LIN {X 0,Y 130.457,Z 414.389,A -85,B 0,C 180,E1 -28269.621,E2 -28269.621} C_VEL
LIN {X 0,Y 125.281,Z 421.79,A -85,B 0,C 180,E1 -28270.976,E2 -28270.976} C_VEL
LIN {X 0,Y 118.932,Z 429.346,A -85,B 0,C 180,E1 -28272.835,E2 -28272.835} C_VEL
LIN {X 0,Y 111.008,Z 437.034,A -85,B 0,C 180,E1 -28275.509,E2 -28275.509} C_VEL
LIN {X 0,Y 103.666,Z 442.686,A -85,B 0,C 180,E1 -28278.357,E2 -28278.357} C_VEL
LIN {X 0,Y 97.893,Z 446.46,A -85,B 0,C 180,E1 -28281.046,E2 -28281.046} C_VEL
LIN {X 0,Y 92.339,Z 449.512,A -85,B 0,C 180,E1 -28284.033,E2 -28284.033} C_VEL
LIN {X 0,Y 87.083,Z 451.866,A -85,B 0,C 180,E1 -28287.41,E2 -28287.41} C_VEL
LIN {X 0,Y 82.167,Z 453.567,A -85,B 0,C 180,E1 -28291.205,E2 -28291.205} C_VEL
LIN {X 0,Y 77.631,Z 454.708,A -85,B 0,C 180,E1 -28295.437,E2 -28295.437} C_VEL
LIN {X 0,Y 71.023,Z 455.494,A -85,B 0,C 180,E1 -28303.815,E2 -28303.815} C_VEL
LIN {X 0,Y 67.098,Z 454.979,A -85,B 0,C 180,E1 -28311.065,E2 -28311.065} C_VEL
LIN {X 0,Y 64.842,Z 453.933,A -85,B 0,C 180,E1 -28317.186,E2 -28317.186} C_VEL
LIN {X 0,Y 62.895,Z 451.358,A -85,B 0,C 180,E1 -28326.979,E2 -28326.979} C_VEL
LIN {X 0,Y 62.503,Z 448.908,A -85,B 0,C 180,E1 -28333.675,E2 -28333.675} C_VEL
LIN {X 0,Y 63.308,Z 443.942,A -85,B 0,C 180,E1 -28343.628,E2 -28343.628} C_VEL
LIN {X 0,Y 65.146,Z 438.567,A -85,B 0,C 180,E1 -28351.547,E2 -28351.547} C_VEL
LIN {X 0,Y 67.153,Z 433.329,A -85,B 0,C 180,E1 -28357.518,E2 -28357.518} C_VEL
LIN {X 0,Y 69.776,Z 427.008,A -85,B 0,C 180,E1 -28363.1,E2 -28363.1} C_VEL
LIN {X 0,Y 72.514,Z 420.358,A -85,B 0,C 180,E1 -28367.631,E2 -28367.631} C_VEL
LIN {X 0,Y 75.671,Z 412.288,A -85,B 0,C 180,E1 -28371.809,E2 -28371.809} C_VEL
LIN {X 0,Y 78.693,Z 403.494,A -85,B 0,C 180,E1 -28375.219,E2 -28375.219} C_VEL
LIN {X 0,Y 81.712,Z 392.43,A -85,B 0,C 180,E1 -28378.324,E2 -28378.324} C_VEL
LIN {X 0,Y 83.873,Z 381.725,A -85,B 0,C 180,E1 -28380.297,E2 -28380.297} C_VEL
LIN {X 0,Y 85.27,Z 372.1,A -85,B 0,C 180,E1 -28381.419,E2 -28381.419} C_VEL
LIN {X 0,Y 87.182,Z 347.964,A -85,B 0,C 180,E1 -28383.17,E2 -28383.17} C_VEL
LIN {X 0,Y 84.324,Z 341.212,A -85,B 0,C 180,E1 -28385.816,E2 -28385.816} C_VEL
LIN {X 0,Y 79.131,Z 331.666,A -85,B 0,C 180,E1 -28391.138,E2 -28391.138} C_VEL
LIN {X 0,Y 75.765,Z 326.616,A -85,B 0,C 180,E1 -28395.162,E2 -28395.162} C_VEL
LIN {X 0,Y 73.243,Z 322.884,A -85,B 0,C 180,E1 -28398.715,E2 -28398.715} C_VEL
LIN {X 0,Y 70.889,Z 320.396,A -85,B 0,C 180,E1 -28402.421,E2 -28402.421} C_VEL
LIN {X 0,Y 69.816,Z 317.967,A -85,B 0,C 180,E1 -28404.656,E2 -28404.656} C_VEL
LIN {X 0,Y 67.219,Z 316.228,A -85,B 0,C 180,E1 -28410.108,E2 -28410.108} C_VEL
LIN {X 0,Y 65.712,Z 313.659,A -85,B 0,C 180,E1 -28414.906,E2 -28414.906} C_VEL
LIN {X 0,Y 65.448,Z 312.106,A -85,B 0,C 180,E1 -28416.696,E2 -28416.696} C_VEL
LIN {X 0,Y 70.33,Z 311.511,A -85,B 0,C 180,E1 -28437.877,E2 -28437.877} C_VEL
LIN {X 0,Y 75.148,Z 311.098,A -85,B 0,C 180,E1 -28444.711,E2 -28444.711} C_VEL
LIN {X 0,Y 80.078,Z 356.507,A -85,B 0,C 180,E1 -28453.675,E2 -28453.675} C_VEL
LIN {X 0,Y 81.204,Z 367.651,A -85,B 0,C 180,E1 -28456.127,E2 -28456.127} C_VEL
LIN {X 0,Y 81.915,Z 377.696,A -85,B 0,C 180,E1 -28459.031,E2 -28459.031} C_VEL
LIN {X 0,Y 82.52,Z 385.251,A -85,B 0,C 180,E1 -28461.893,E2 -28461.893} C_VEL
LIN {X 0,Y 83.392,Z 393.266,A -85,B 0,C 180,E1 -28465.969,E2 -28465.969} C_VEL
LIN {X 0,Y 84.869,Z 401.147,A -85,B 0,C 180,E1 -28470.72,E2 -28470.72} C_VEL
LIN {X 0,Y 87.441,Z 409.064,A -85,B 0,C 180,E1 -28475.939,E2 -28475.939} C_VEL
LIN {X 0,Y 93.038,Z 419.345,A -85,B 0,C 180,E1 -28482.849,E2 -28482.849} C_VEL
LIN {X 0,Y 94.672,Z 421.602,A -85,B 0,C 180,E1 -28484.351,E2 -28484.351} C_VEL
LIN {X 0,Y 93.114,Z 419.795,A -85,B 0,C 180,E1 -28487.21,E2 -28487.21} C_VEL
LIN {X 0,Y 88.882,Z 413.219,A -85,B 0,C 180,E1 -28493.557,E2 -28493.557} C_VEL
LIN {X 0,Y 84.438,Z 418.04,A -85,B 0,C 180,E1 -28494.363,E2 -28494.363} C_VEL
LIN {X 0,Y 79.435,Z 424.487,A -85,B 0,C 180,E1 -28496.428,E2 -28496.428} C_VEL
LIN {X 0,Y 74.169,Z 431.806,A -85,B 0,C 180,E1 -28500.166,E2 -28500.166} C_VEL
LIN {X 0,Y 70.273,Z 437.549,A -85,B 0,C 180,E1 -28504.351,E2 -28504.351} C_VEL
LIN {X 0,Y 66.983,Z 443.216,A -85,B 0,C 180,E1 -28510.061,E2 -28510.061} C_VEL
LIN {X 0,Y 64.441,Z 448.562,A -85,B 0,C 180,E1 -28517.4,E2 -28517.4} C_VEL
LIN {X 0,Y 63.41,Z 452.058,A -85,B 0,C 180,E1 -28523.635,E2 -28523.635} C_VEL
LIN {X 0,Y 63.272,Z 454.934,A -85,B 0,C 180,E1 -28529.999,E2 -28529.999} C_VEL
LIN {X 0,Y 63.085,Z 457.125,A -85,B 0,C 180,E1 -28536.395,E2 -28536.395} C_VEL
LIN {X 0,Y 63.598,Z 458.696,A -85,B 0,C 180,E1 -28542.767,E2 -28542.767} C_VEL
LIN {X 0,Y 64.839,Z 459.786,A -85,B 0,C 180,E1 -28548.975,E2 -28548.975} C_VEL
LIN {X 0,Y 66.817,Z 460.43,A -85,B 0,C 180,E1 -28554.879,E2 -28554.879} C_VEL
LIN {X 0,Y 69.423,Z 460.623,A -85,B 0,C 180,E1 -28560.408,E2 -28560.408} C_VEL
LIN {X 0,Y 72.698,Z 460.247,A -85,B 0,C 180,E1 -28565.452,E2 -28565.452} C_VEL
LIN {X 0,Y 76.592,Z 459.396,A -85,B 0,C 180,E1 -28569.963,E2 -28569.963} C_VEL
LIN {X 0,Y 80.924,Z 458.092,A -85,B 0,C 180,E1 -28574.008,E2 -28574.008} C_VEL
LIN {X 0,Y 88.109,Z 455.143,A -85,B 0,C 180,E1 -28579.267,E2 -28579.267} C_VEL
LIN {X 0,Y 93.327,Z 452.493,A -85,B 0,C 180,E1 -28582.25,E2 -28582.25} C_VEL
LIN {X 0,Y 101.608,Z 447.322,A -85,B 0,C 180,E1 -28586.099,E2 -28586.099} C_VEL
LIN {X 0,Y 109.921,Z 440.844,A -85,B 0,C 180,E1 -28589.31,E2 -28589.31} C_VEL
LIN {X 0,Y 117.751,Z 433.257,A -85,B 0,C 180,E1 -28591.685,E2 -28591.685} C_VEL
LIN {X 0,Y 123.906,Z 426.049,A -85,B 0,C 180,E1 -28593.296,E2 -28593.296} C_VEL
LIN {X 0,Y 129.407,Z 418.363,A -85,B 0,C 180,E1 -28594.54,E2 -28594.54} C_VEL
LIN {X 0,Y 133.967,Z 410.731,A -85,B 0,C 180,E1 -28595.444,E2 -28595.444} C_VEL
LIN {X 0,Y 138.255,Z 401.917,A -85,B 0,C 180,E1 -28596.205,E2 -28596.205} C_VEL
LIN {X 0,Y 139.851,Z 398.143,A -85,B 0,C 180,E1 -28596.509,E2 -28596.509} C_VEL
LIN {X 0,Y 139.681,Z 393.765,A -85,B 0,C 180,E1 -28599.369,E2 -28599.369} C_VEL
LIN {X 0,Y 139.428,Z 392.17,A -85,B 0,C 180,E1 -28600.927,E2 -28600.927} C_VEL
LIN {X 0,Y 138.957,Z 389.849,A -85,B 0,C 180,E1 -28603.935,E2 -28603.935} C_VEL
LIN {X 0,Y 138.331,Z 386.897,A -85,B 0,C 180,E1 -28611.224,E2 -28611.224} C_VEL
LIN {X 0,Y 138.451,Z 386.702,A -85,B 0,C 180,E1 -28614.164,E2 -28614.164} C_VEL
LIN {X 0,Y 138.714,Z 389.539,A -85,B 0,C 180,E1 -28619.991,E2 -28619.991} C_VEL
LIN {X 0,Y 139.208,Z 393.208,A -85,B 0,C 180,E1 -28624.334,E2 -28624.334} C_VEL
LIN {X 0,Y 139.334,Z 394.063,A -85,B 0,C 180,E1 -28625.176,E2 -28625.176} C_VEL
LIN {X 0,Y 139.116,Z 395.586,A -85,B 0,C 180,E1 -28625.911,E2 -28625.911} C_VEL
LIN {X 0,Y 138.136,Z 398.315,A -85,B 0,C 180,E1 -28626.389,E2 -28626.389} C_VEL
LIN {X 0,Y 136.101,Z 402.524,A -85,B 0,C 180,E1 -28626.493,E2 -28626.493} C_VEL
LIN {X 0,Y 131.283,Z 410.331,A -85,B 0,C 180,E1 -28626.163,E2 -28626.163} C_VEL
LIN {X 0,Y 129.637,Z 412.827,A -85,B 0,C 180,E1 -28626.35,E2 -28626.35} C_VEL
LIN {X 0,Y 124.077,Z 420.81,A -85,B 0,C 180,E1 -28627.595,E2 -28627.595} C_VEL
LIN {X 0,Y 119.137,Z 426.82,A -85,B 0,C 180,E1 -28628.854,E2 -28628.854} C_VEL
LIN {X 0,Y 112.163,Z 433.882,A -85,B 0,C 180,E1 -28630.823,E2 -28630.823} C_VEL
LIN {X 0,Y 104.693,Z 440.112,A -85,B 0,C 180,E1 -28633.254,E2 -28633.254} C_VEL
LIN {X 0,Y 98.493,Z 444.382,A -85,B 0,C 180,E1 -28635.575,E2 -28635.575} C_VEL
LIN {X 0,Y 92.028,Z 448.107,A -85,B 0,C 180,E1 -28638.443,E2 -28638.443} C_VEL
LIN {X 0,Y 83.908,Z 451.828,A -85,B 0,C 180,E1 -28642.879,E2 -28642.879} C_VEL
LIN {X 0,Y 78.468,Z 453.66,A -85,B 0,C 180,E1 -28646.585,E2 -28646.585} C_VEL
LIN {X 0,Y 73.547,Z 454.886,A -85,B 0,C 180,E1 -28650.684,E2 -28650.684} C_VEL
LIN {X 0,Y 68.987,Z 455.606,A -85,B 0,C 180,E1 -28655.415,E2 -28655.415} C_VEL
LIN {X 0,Y 64.945,Z 455.807,A -85,B 0,C 180,E1 -28660.758,E2 -28660.758} C_VEL
LIN {X 0,Y 61.48,Z 455.417,A -85,B 0,C 180,E1 -28666.696,E2 -28666.696} C_VEL
LIN {X 0,Y 58.722,Z 454.44,A -85,B 0,C 180,E1 -28673.245,E2 -28673.245} C_VEL
LIN {X 0,Y 56.128,Z 452.049,A -85,B 0,C 180,E1 -28684.009,E2 -28684.009} C_VEL
LIN {X 0,Y 55.418,Z 448.224,A -85,B 0,C 180,E1 -28695.309,E2 -28695.309} C_VEL
LIN {X 0,Y 56.395,Z 443.599,A -85,B 0,C 180,E1 -28705.23,E2 -28705.23} C_VEL
LIN {X 0,Y 58.367,Z 438.473,A -85,B 0,C 180,E1 -28713.453,E2 -28713.453} C_VEL
LIN {X 0,Y 60.615,Z 433.152,A -85,B 0,C 180,E1 -28720.017,E2 -28720.017} C_VEL
LIN {X 0,Y 63.546,Z 426.73,A -85,B 0,C 180,E1 -28726.052,E2 -28726.052} C_VEL
LIN {X 0,Y 67.556,Z 417.869,A -85,B 0,C 180,E1 -28732.156,E2 -28732.156} C_VEL
LIN {X 0,Y 71.497,Z 407.795,A -85,B 0,C 180,E1 -28736.947,E2 -28736.947} C_VEL
LIN {X 0,Y 74.353,Z 399.47,A -85,B 0,C 180,E1 -28739.753,E2 -28739.753} C_VEL
LIN {X 0,Y 76.853,Z 390.146,A -85,B 0,C 180,E1 -28742.111,E2 -28742.111} C_VEL
LIN {X 0,Y 78.787,Z 380.756,A -85,B 0,C 180,E1 -28743.772,E2 -28743.772} C_VEL
LIN {X 0,Y 80.185,Z 371.132,A -85,B 0,C 180,E1 -28744.848,E2 -28744.848} C_VEL
LIN {X 0,Y 81.93,Z 350.008,A -85,B 0,C 180,E1 -28746.413,E2 -28746.413} C_VEL
LIN {X 0,Y 79.46,Z 344.241,A -85,B 0,C 180,E1 -28749.083,E2 -28749.083} C_VEL
LIN {X 0,Y 75.348,Z 336.338,A -85,B 0,C 180,E1 -28754.021,E2 -28754.021} C_VEL
LIN {X 0,Y 72.573,Z 332.018,A -85,B 0,C 180,E1 -28757.856,E2 -28757.856} C_VEL
LIN {X 0,Y 70.65,Z 329.013,A -85,B 0,C 180,E1 -28760.957,E2 -28760.957} C_VEL
LIN {X 0,Y 68.282,Z 325.962,A -85,B 0,C 180,E1 -28765.357,E2 -28765.357} C_VEL
LIN {X 0,Y 67.655,Z 324.536,A -85,B 0,C 180,E1 -28766.865,E2 -28766.865} C_VEL
LIN {X 0,Y 65.267,Z 322.375,A -85,B 0,C 180,E1 -28772.878,E2 -28772.878} C_VEL
LIN {X 0,Y 64.053,Z 319.715,A -85,B 0,C 180,E1 -28777.864,E2 -28777.864} C_VEL
LIN {X 0,Y 63.854,Z 318.969,A -85,B 0,C 180,E1 -28779.063,E2 -28779.063} C_VEL
LIN {X 0,Y 62.674,Z 317.487,A -85,B 0,C 180,E1 -28789.522,E2 -28789.522} C_VEL
LIN {X 0,Y 63.268,Z 315.101,A -85,B 0,C 180,E1 -28796.991,E2 -28796.991} C_VEL
LIN {X 0,Y 64.046,Z 312.858,A -85,B 0,C 180,E1 -28800.413,E2 -28800.413} C_VEL
LIN {X 0,Y 64.388,Z 312.272,A -85,B 0,C 180,E1 -28801.193,E2 -28801.193} C_VEL
LIN {X 0,Y 70.156,Z 311.553,A -85,B 0,C 180,E1 -28808.661,E2 -28808.661} C_VEL
LIN {X 0,Y 75.977,Z 356.93,A -85,B 0,C 180,E1 -28818.034,E2 -28818.034} C_VEL
LIN {X 0,Y 77.242,Z 367.844,A -85,B 0,C 180,E1 -28820.612,E2 -28820.612} C_VEL
LIN {X 0,Y 78.05,Z 376.177,A -85,B 0,C 180,E1 -28823.217,E2 -28823.217} C_VEL
LIN {X 0,Y 78.768,Z 382.764,A -85,B 0,C 180,E1 -28825.801,E2 -28825.801} C_VEL
LIN {X 0,Y 80.176,Z 392.373,A -85,B 0,C 180,E1 -28830.941,E2 -28830.941} C_VEL
LIN {X 0,Y 82.567,Z 401.252,A -85,B 0,C 180,E1 -28836.59,E2 -28836.59} C_VEL
LIN {X 0,Y 87.688,Z 412.169,A -85,B 0,C 180,E1 -28843.834,E2 -28843.834} C_VEL
LIN {X 0,Y 89.092,Z 414.368,A -85,B 0,C 180,E1 -28845.25,E2 -28845.25} C_VEL
LIN {X 0,Y 85.771,Z 408.902,A -85,B 0,C 180,E1 -28850.45,E2 -28850.45} C_VEL
LIN {X 0,Y 81.591,Z 413.122,A -85,B 0,C 180,E1 -28850.849,E2 -28850.849} C_VEL
LIN {X 0,Y 77.065,Z 418.627,A -85,B 0,C 180,E1 -28852.005,E2 -28852.005} C_VEL
LIN {X 0,Y 72.249,Z 424.988,A -85,B 0,C 180,E1 -28854.291,E2 -28854.291} C_VEL
LIN {X 0,Y 66.949,Z 432.195,A -85,B 0,C 180,E1 -28858.338,E2 -28858.338} C_VEL
LIN {X 0,Y 63.263,Z 437.614,A -85,B 0,C 180,E1 -28862.755,E2 -28862.755} C_VEL
LIN {X 0,Y 59.702,Z 443.409,A -85,B 0,C 180,E1 -28869.318,E2 -28869.318} C_VEL
LIN {X 0,Y 57.58,Z 447.722,A -85,B 0,C 180,E1 -28875.869,E2 -28875.869} C_VEL
LIN {X 0,Y 56.195,Z 452.827,A -85,B 0,C 180,E1 -28886.413,E2 -28886.413} C_VEL
LIN {X 0,Y 56.205,Z 454.283,A -85,B 0,C 180,E1 -28889.999,E2 -28889.999} C_VEL
LIN {X 0,Y 56.055,Z 456.497,A -85,B 0,C 180,E1 -28897.201,E2 -28897.201} C_VEL
LIN {X 0,Y 56.695,Z 458.149,A -85,B 0,C 180,E1 -28904.353,E2 -28904.353} C_VEL
LIN {X 0,Y 58.16,Z 459.327,A -85,B 0,C 180,E1 -28911.254,E2 -28911.254} C_VEL
LIN {X 0,Y 60.43,Z 460.057,A -85,B 0,C 180,E1 -28917.722,E2 -28917.722} C_VEL
LIN {X 0,Y 63.382,Z 460.289,A -85,B 0,C 180,E1 -28923.669,E2 -28923.669} C_VEL
LIN {X 0,Y 67.041,Z 459.963,A -85,B 0,C 180,E1 -28928.974,E2 -28928.974} C_VEL
LIN {X 0,Y 71.296,Z 459.199,A -85,B 0,C 180,E1 -28933.631,E2 -28933.631} C_VEL
LIN {X 0,Y 75.966,Z 457.983,A -85,B 0,C 180,E1 -28937.74,E2 -28937.74} C_VEL
LIN {X 0,Y 83.656,Z 455.131,A -85,B 0,C 180,E1 -28942.948,E2 -28942.948} C_VEL
LIN {X 0,Y 92.002,Z 451.056,A -85,B 0,C 180,E1 -28947.169,E2 -28947.169} C_VEL
LIN {X 0,Y 100.766,Z 445.605,A -85,B 0,C 180,E1 -28950.67,E2 -28950.67} C_VEL
LIN {X 0,Y 108.352,Z 439.686,A -85,B 0,C 180,E1 -28953.107,E2 -28953.107} C_VEL
LIN {X 0,Y 116.145,Z 432.213,A -85,B 0,C 180,E1 -28955.182,E2 -28955.182} C_VEL
LIN {X 0,Y 122.5,Z 424.864,A -85,B 0,C 180,E1 -28956.626,E2 -28956.626} C_VEL
LIN {X 0,Y 128.153,Z 417.003,A -85,B 0,C 180,E1 -28957.732,E2 -28957.732} C_VEL
LIN {X 0,Y 133.325,Z 408.252,A -85,B 0,C 180,E1 -28958.596,E2 -28958.596} C_VEL
LIN {X 0,Y 136.379,Z 401.889,A -85,B 0,C 180,E1 -28959.07,E2 -28959.07} C_VEL
LIN {X 0,Y 136.676,Z 399.651,A -85,B 0,C 180,E1 -28960.463,E2 -28960.463} C_VEL
LIN {X 0,Y 136.418,Z 397.023,A -85,B 0,C 180,E1 -28963.627,E2 -28963.627} C_VEL
LIN {X 0,Y 136.274,Z 396.091,A -85,B 0,C 180,E1 -28965.047,E2 -28965.047} C_VEL
LIN {X 0,Y 135.969,Z 393.72,A -85,B 0,C 180,E1 -28971.07,E2 -28971.07} C_VEL
LIN {X 0,Y 136.066,Z 393.495,A -85,B 0,C 180,E1 -28974.061,E2 -28974.061} C_VEL
LIN {X 0,Y 136.064,Z 396.477,A -85,B 0,C 180,E1 -28979.99,E2 -28979.99} C_VEL
LIN {X 0,Y 136.138,Z 400.277,A -85,B 0,C 180,E1 -28984.58,E2 -28984.58} C_VEL
LIN {X 0,Y 136.146,Z 400.62,A -85,B 0,C 180,E1 -28984.913,E2 -28984.913} C_VEL
LIN {X 0,Y 131.331,Z 410.103,A -85,B 0,C 180,E1 -28985.99,E2 -28985.99} C_VEL
LIN {X 0,Y 129.637,Z 412.827,A -85,B 0,C 180,E1 -28986.35,E2 -28986.35} C_VEL
LIN {X 0,Y 126.256,Z 417.745,A -85,B 0,C 180,E1 -28986.767,E2 -28986.767} C_VEL
LIN {X 0,Y 119.636,Z 425.325,A -85,B 0,C 180,E1 -28986.795,E2 -28986.795} C_VEL
LIN {X 0,Y 112.539,Z 432.075,A -85,B 0,C 180,E1 -28987.002,E2 -28987.002} C_VEL
LIN {X 0,Y 108.327,Z 435.68,A -85,B 0,C 180,E1 -28987.775,E2 -28987.775} C_VEL
LIN {X 0,Y 99.979,Z 442.094,A -85,B 0,C 180,E1 -28990.226,E2 -28990.226} C_VEL
LIN {X 0,Y 91.444,Z 447.21,A -85,B 0,C 180,E1 -28993.315,E2 -28993.315} C_VEL
LIN {X 0,Y 84.276,Z 450.622,A -85,B 0,C 180,E1 -28996.462,E2 -28996.462} C_VEL
LIN {X 0,Y 74.432,Z 454.03,A -85,B 0,C 180,E1 -29002.171,E2 -29002.171} C_VEL
LIN {X 0,Y 70.021,Z 455.074,A -85,B 0,C 180,E1 -29005.404,E2 -29005.404} C_VEL
LIN {X 0,Y 64.941,Z 455.898,A -85,B 0,C 180,E1 -29010.031,E2 -29010.031} C_VEL
LIN {X 0,Y 59.94,Z 456.158,A -85,B 0,C 180,E1 -29015.863,E2 -29015.863} C_VEL
LIN {X 0,Y 56.28,Z 455.815,A -85,B 0,C 180,E1 -29021.476,E2 -29021.476} C_VEL
LIN {X 0,Y 52.936,Z 454.945,A -85,B 0,C 180,E1 -29028.41,E2 -29028.41} C_VEL
LIN {X 0,Y 50.205,Z 453.344,A -85,B 0,C 180,E1 -29037.081,E2 -29037.081} C_VEL
LIN {X 0,Y 48.504,Z 450.38,A -85,B 0,C 180,E1 -29048.764,E2 -29048.764} C_VEL
LIN {X 0,Y 48.755,Z 445.867,A -85,B 0,C 180,E1 -29061.714,E2 -29061.714} C_VEL
LIN {X 0,Y 50.576,Z 440.812,A -85,B 0,C 180,E1 -29071.992,E2 -29071.992} C_VEL
LIN {X 0,Y 53.542,Z 434.424,A -85,B 0,C 180,E1 -29081.357,E2 -29081.357} C_VEL
LIN {X 0,Y 56.637,Z 428.197,A -85,B 0,C 180,E1 -29088.074,E2 -29088.074} C_VEL
LIN {X 0,Y 59.938,Z 421.64,A -85,B 0,C 180,E1 -29093.313,E2 -29093.313} C_VEL
LIN {X 0,Y 63.183,Z 414.694,A -85,B 0,C 180,E1 -29097.502,E2 -29097.502} C_VEL
LIN {X 0,Y 66.232,Z 407.319,A -85,B 0,C 180,E1 -29100.892,E2 -29100.892} C_VEL
LIN {X 0,Y 68.817,Z 400.372,A -85,B 0,C 180,E1 -29103.295,E2 -29103.295} C_VEL
LIN {X 0,Y 71.465,Z 391.239,A -85,B 0,C 180,E1 -29105.727,E2 -29105.727} C_VEL
LIN {X 0,Y 73.636,Z 381.781,A -85,B 0,C 180,E1 -29107.434,E2 -29107.434} C_VEL
LIN {X 0,Y 75.176,Z 372.245,A -85,B 0,C 180,E1 -29108.529,E2 -29108.529} C_VEL
LIN {X 0,Y 76.972,Z 352.143,A -85,B 0,C 180,E1 -29110.079,E2 -29110.079} C_VEL
LIN {X 0,Y 73.015,Z 343.412,A -85,B 0,C 180,E1 -29115.331,E2 -29115.331} C_VEL
LIN {X 0,Y 69.63,Z 337.529,A -85,B 0,C 180,E1 -29120.639,E2 -29120.639} C_VEL
LIN {X 0,Y 68.047,Z 334.961,A -85,B 0,C 180,E1 -29123.6,E2 -29123.6} C_VEL
LIN {X 0,Y 65.774,Z 331.311,A -85,B 0,C 180,E1 -29128.778,E2 -29128.778} C_VEL
LIN {X 0,Y 63.04,Z 327.611,A -85,B 0,C 180,E1 -29137.813,E2 -29137.813} C_VEL
LIN {X 0,Y 62.539,Z 325.828,A -85,B 0,C 180,E1 -29141.11,E2 -29141.11} C_VEL
LIN {X 0,Y 61.815,Z 324.122,A -85,B 0,C 180,E1 -29151.851,E2 -29151.851} C_VEL
LIN {X 0,Y 62.803,Z 321.557,A -85,B 0,C 180,E1 -29159.64,E2 -29159.64} C_VEL
LIN {X 0,Y 64.008,Z 319.003,A -85,B 0,C 180,E1 -29163.953,E2 -29163.953} C_VEL
LIN {X 0,Y 64.879,Z 318.49,A -85,B 0,C 180,E1 -29166.824,E2 -29166.824} C_VEL
LIN {X 0,Y 65.14,Z 329.275,A -85,B 0,C 180,E1 -29171.494,E2 -29171.494} C_VEL
LIN {X 0,Y 65.779,Z 333.915,A -85,B 0,C 180,E1 -29174.316,E2 -29174.316} C_VEL
LIN {X 0,Y 66.257,Z 335.047,A -85,B 0,C 180,E1 -29175.582,E2 -29175.582} C_VEL
LIN {X 0,Y 66.769,Z 334.861,A -85,B 0,C 180,E1 -29176.494,E2 -29176.494} C_VEL
LIN {X 0,Y 67.367,Z 332.904,A -85,B 0,C 180,E1 -29177.078,E2 -29177.078} C_VEL
LIN {X 0,Y 67.851,Z 329.395,A -85,B 0,C 180,E1 -29177.062,E2 -29177.062} C_VEL
LIN {X 0,Y 72.311,Z 356.278,A -85,B 0,C 180,E1 -29182.734,E2 -29182.734} C_VEL
LIN {X 0,Y 73.954,Z 367.504,A -85,B 0,C 180,E1 -29185.525,E2 -29185.525} C_VEL
LIN {X 0,Y 75.118,Z 376.804,A -85,B 0,C 180,E1 -29188.671,E2 -29188.671} C_VEL
LIN {X 0,Y 76.088,Z 384.013,A -85,B 0,C 180,E1 -29192.099,E2 -29192.099} C_VEL
LIN {X 0,Y 78.185,Z 392.918,A -85,B 0,C 180,E1 -29197.373,E2 -29197.373} C_VEL
LIN {X 0,Y 82.43,Z 403.63,A -85,B 0,C 180,E1 -29204.39,E2 -29204.39} C_VEL
LIN {X 0,Y 83.1,Z 404.894,A -85,B 0,C 180,E1 -29205.192,E2 -29205.192} C_VEL
LIN {X 0,Y 82.699,Z 404.297,A -85,B 0,C 180,E1 -29207.429,E2 -29207.429} C_VEL
LIN {X 0,Y 78.275,Z 408.962,A -85,B 0,C 180,E1 -29207.337,E2 -29207.337} C_VEL
LIN {X 0,Y 72.631,Z 415.885,A -85,B 0,C 180,E1 -29208.297,E2 -29208.297} C_VEL
LIN {X 0,Y 66.736,Z 423.585,A -85,B 0,C 180,E1 -29210.811,E2 -29210.811} C_VEL
LIN {X 0,Y 61.108,Z 430.962,A -85,B 0,C 180,E1 -29214.896,E2 -29214.896} C_VEL
LIN {X 0,Y 56.642,Z 437.197,A -85,B 0,C 180,E1 -29220.242,E2 -29220.242} C_VEL
LIN {X 0,Y 53.184,Z 442.454,A -85,B 0,C 180,E1 -29226.643,E2 -29226.643} C_VEL
LIN {X 0,Y 50.762,Z 446.88,A -85,B 0,C 180,E1 -29233.923,E2 -29233.923} C_VEL
LIN {X 0,Y 49.393,Z 450.583,A -85,B 0,C 180,E1 -29241.818,E2 -29241.818} C_VEL
LIN {X 0,Y 49.127,Z 453.589,A -85,B 0,C 180,E1 -29249.998,E2 -29249.998} C_VEL
LIN {X 0,Y 49.054,Z 455.86,A -85,B 0,C 180,E1 -29258.236,E2 -29258.236} C_VEL
LIN {X 0,Y 49.858,Z 457.603,A -85,B 0,C 180,E1 -29266.373,E2 -29266.373} C_VEL
LIN {X 0,Y 51.604,Z 458.869,A -85,B 0,C 180,E1 -29274.114,E2 -29274.114} C_VEL
LIN {X 0,Y 54.232,Z 459.679,A -85,B 0,C 180,E1 -29281.221,E2 -29281.221} C_VEL
LIN {X 0,Y 57.592,Z 459.921,A -85,B 0,C 180,E1 -29287.599,E2 -29287.599} C_VEL
LIN {X 0,Y 61.687,Z 459.68,A -85,B 0,C 180,E1 -29293.123,E2 -29293.123} C_VEL
LIN {X 0,Y 66.339,Z 459.008,A -85,B 0,C 180,E1 -29297.865,E2 -29297.865} C_VEL
LIN {X 0,Y 71.376,Z 457.888,A -85,B 0,C 180,E1 -29301.971,E2 -29301.971} C_VEL
LIN {X 0,Y 79.588,Z 455.138,A -85,B 0,C 180,E1 -29307.022,E2 -29307.022} C_VEL
LIN {X 0,Y 88.353,Z 451.169,A -85,B 0,C 180,E1 -29311.042,E2 -29311.042} C_VEL
LIN {X 0,Y 94.433,Z 447.762,A -85,B 0,C 180,E1 -29313.261,E2 -29313.261} C_VEL
LIN {X 0,Y 102.166,Z 442.495,A -85,B 0,C 180,E1 -29315.707,E2 -29315.707} C_VEL
LIN {X 0,Y 108.538,Z 437.345,A -85,B 0,C 180,E1 -29317.324,E2 -29317.324} C_VEL
LIN {X 0,Y 114.974,Z 431.172,A -85,B 0,C 180,E1 -29318.776,E2 -29318.776} C_VEL
LIN {X 0,Y 120.691,Z 424.698,A -85,B 0,C 180,E1 -29319.88,E2 -29319.88} C_VEL
LIN {X 0,Y 126.482,Z 416.867,A -85,B 0,C 180,E1 -29320.839,E2 -29320.839} C_VEL
LIN {X 0,Y 131.793,Z 408.081,A -85,B 0,C 180,E1 -29321.598,E2 -29321.598} C_VEL
LIN {X 0,Y 133.189,Z 405.532,A -85,B 0,C 180,E1 -29321.769,E2 -29321.769} C_VEL
LIN {X 0,Y 133.336,Z 404.016,A -85,B 0,C 180,E1 -29323.137,E2 -29323.137} C_VEL
LIN {X 0,Y 133.273,Z 402.921,A -85,B 0,C 180,E1 -29324.703,E2 -29324.703} C_VEL
LIN {X 0,Y 133.129,Z 400.436,A -85,B 0,C 180,E1 -29330.878,E2 -29330.878} C_VEL
LIN {X 0,Y 133.25,Z 400.082,A -85,B 0,C 180,E1 -29333.935,E2 -29333.935} C_VEL
LIN {X 0,Y 132.908,Z 403.136,A -85,B 0,C 180,E1 -29339.99,E2 -29339.99} C_VEL
LIN {X 0,Y 132.744,Z 404.85,A -85,B 0,C 180,E1 -29342.267,E2 -29342.267} C_VEL
LIN {X 0,Y 131.255,Z 407.626,A -85,B 0,C 180,E1 -29342.664,E2 -29342.664} C_VEL
LIN {X 0,Y 125.882,Z 416.262,A -85,B 0,C 180,E1 -29343.664,E2 -29343.664} C_VEL
LIN {X 0,Y 119.919,Z 424.086,A -85,B 0,C 180,E1 -29344.931,E2 -29344.931} C_VEL
LIN {X 0,Y 113.176,Z 431.347,A -85,B 0,C 180,E1 -29346.507,E2 -29346.507} C_VEL
LIN {X 0,Y 108.327,Z 435.68,A -85,B 0,C 180,E1 -29347.775,E2 -29347.775} C_VEL
LIN {X 0,Y 105.283,Z 438.116,A -85,B 0,C 180,E1 -29348.246,E2 -29348.246} C_VEL
LIN {X 0,Y 99.597,Z 441.771,A -85,B 0,C 180,E1 -29348.102,E2 -29348.102} C_VEL
LIN {X 0,Y 93.677,Z 445.056,A -85,B 0,C 180,E1 -29347.983,E2 -29347.983} C_VEL
LIN {X 0,Y 90.269,Z 446.858,A -85,B 0,C 180,E1 -29348.611,E2 -29348.611} C_VEL
LIN {X 0,Y 82.478,Z 450.591,A -85,B 0,C 180,E1 -29351.506,E2 -29351.506} C_VEL
LIN {X 0,Y 73.109,Z 453.797,A -85,B 0,C 180,E1 -29355.994,E2 -29355.994} C_VEL
LIN {X 0,Y 67.161,Z 455.26,A -85,B 0,C 180,E1 -29359.648,E2 -29359.648} C_VEL
LIN {X 0,Y 61.535,Z 456.172,A -85,B 0,C 180,E1 -29363.982,E2 -29363.982} C_VEL
LIN {X 0,Y 54.94,Z 456.487,A -85,B 0,C 180,E1 -29370.748,E2 -29370.748} C_VEL
LIN {X 0,Y 47.621,Z 455.443,A -85,B 0,C 180,E1 -29382.449,E2 -29382.449} C_VEL
LIN {X 0,Y 43.684,Z 453.627,A -85,B 0,C 180,E1 -29393.5,E2 -29393.5} C_VEL
LIN {X 0,Y 41.684,Z 451.092,A -85,B 0,C 180,E1 -29405.073,E2 -29405.073} C_VEL
LIN {X 0,Y 41.228,Z 448.311,A -85,B 0,C 180,E1 -29415.187,E2 -29415.187} C_VEL
LIN {X 0,Y 42.208,Z 444.199,A -85,B 0,C 180,E1 -29426.835,E2 -29426.835} C_VEL
LIN {X 0,Y 44.435,Z 439.471,A -85,B 0,C 180,E1 -29436.814,E2 -29436.814} C_VEL
LIN {X 0,Y 47.236,Z 434.214,A -85,B 0,C 180,E1 -29445.094,E2 -29445.094} C_VEL
LIN {X 0,Y 50.778,Z 427.882,A -85,B 0,C 180,E1 -29452.374,E2 -29452.374} C_VEL
LIN {X 0,Y 54.467,Z 421.205,A -85,B 0,C 180,E1 -29457.889,E2 -29457.889} C_VEL
LIN {X 0,Y 58.505,Z 413.184,A -85,B 0,C 180,E1 -29462.672,E2 -29462.672} C_VEL
LIN {X 0,Y 62.963,Z 402.986,A -85,B 0,C 180,E1 -29466.869,E2 -29466.869} C_VEL
LIN {X 0,Y 66.498,Z 392.073,A -85,B 0,C 180,E1 -29469.904,E2 -29469.904} C_VEL
LIN {X 0,Y 68.919,Z 382.191,A -85,B 0,C 180,E1 -29471.711,E2 -29471.711} C_VEL
LIN {X 0,Y 70.6,Z 372.517,A -85,B 0,C 180,E1 -29472.784,E2 -29472.784} C_VEL
LIN {X 0,Y 72.342,Z 354.689,A -85,B 0,C 180,E1 -29474.153,E2 -29474.153} C_VEL
LIN {X 0,Y 69.012,Z 346.993,A -85,B 0,C 180,E1 -29479.561,E2 -29479.561} C_VEL
LIN {X 0,Y 65.986,Z 341.335,A -85,B 0,C 180,E1 -29485.61,E2 -29485.61} C_VEL
LIN {X 0,Y 63.597,Z 337.346,A -85,B 0,C 180,E1 -29492.001,E2 -29492.001} C_VEL
LIN {X 0,Y 61.628,Z 333.965,A -85,B 0,C 180,E1 -29500.419,E2 -29500.419} C_VEL
LIN {X 0,Y 61.324,Z 332.692,A -85,B 0,C 180,E1 -29503.118,E2 -29503.118} C_VEL
LIN {X 0,Y 61.058,Z 330.786,A -85,B 0,C 180,E1 -29514.251,E2 -29514.251} C_VEL
LIN {X 0,Y 62.468,Z 328.005,A -85,B 0,C 180,E1 -29522.311,E2 -29522.311} C_VEL
LIN {X 0,Y 62.866,Z 327.318,A -85,B 0,C 180,E1 -29523.69,E2 -29523.69} C_VEL
LIN {X 0,Y 62.997,Z 335.729,A -85,B 0,C 180,E1 -29528.037,E2 -29528.037} C_VEL
LIN {X 0,Y 63.702,Z 340.13,A -85,B 0,C 180,E1 -29531.555,E2 -29531.555} C_VEL
LIN {X 0,Y 64.717,Z 341.838,A -85,B 0,C 180,E1 -29534.373,E2 -29534.373} C_VEL
LIN {X 0,Y 65.051,Z 342.168,A -85,B 0,C 180,E1 -29535.15,E2 -29535.15} C_VEL
LIN {X 0,Y 66.24,Z 361.269,A -85,B 0,C 180,E1 -29541.819,E2 -29541.819} C_VEL
LIN {X 0,Y 68.211,Z 378.087,A -85,B 0,C 180,E1 -29548.017,E2 -29548.017} C_VEL
LIN {X 0,Y 69.235,Z 385.547,A -85,B 0,C 180,E1 -29551.369,E2 -29551.369} C_VEL
LIN {X 0,Y 70.865,Z 393.104,A -85,B 0,C 180,E1 -29555.658,E2 -29555.658} C_VEL
LIN {X 0,Y 73.227,Z 400.417,A -85,B 0,C 180,E1 -29560.496,E2 -29560.496} C_VEL
LIN {X 0,Y 75.101,Z 404.695,A -85,B 0,C 180,E1 -29563.661,E2 -29563.661} C_VEL
LIN {X 0,Y 69.833,Z 411.228,A -85,B 0,C 180,E1 -29564.003,E2 -29564.003} C_VEL
LIN {X 0,Y 64.883,Z 417.631,A -85,B 0,C 180,E1 -29565.244,E2 -29565.244} C_VEL
LIN {X 0,Y 59.917,Z 424.092,A -85,B 0,C 180,E1 -29567.587,E2 -29567.587} C_VEL
LIN {X 0,Y 54.28,Z 431.34,A -85,B 0,C 180,E1 -29571.998,E2 -29571.998} C_VEL
LIN {X 0,Y 49.65,Z 437.503,A -85,B 0,C 180,E1 -29577.937,E2 -29577.937} C_VEL
LIN {X 0,Y 46.057,Z 442.659,A -85,B 0,C 180,E1 -29585.187,E2 -29585.187} C_VEL
LIN {X 0,Y 43.066,Z 447.927,A -85,B 0,C 180,E1 -29595.829,E2 -29595.829} C_VEL
LIN {X 0,Y 42.084,Z 451.354,A -85,B 0,C 180,E1 -29605.208,E2 -29605.208} C_VEL
LIN {X 0,Y 42.059,Z 452.856,A -85,B 0,C 180,E1 -29609.998,E2 -29609.998} C_VEL
LIN {X 0,Y 42.056,Z 455.216,A -85,B 0,C 180,E1 -29619.618,E2 -29619.618} C_VEL
LIN {X 0,Y 43.09,Z 457.048,A -85,B 0,C 180,E1 -29629.036,E2 -29629.036} C_VEL
LIN {X 0,Y 45.22,Z 458.404,A -85,B 0,C 180,E1 -29637.789,E2 -29637.789} C_VEL
LIN {X 0,Y 48.294,Z 459.261,A -85,B 0,C 180,E1 -29645.597,E2 -29645.597} C_VEL
LIN {X 0,Y 52.135,Z 459.547,A -85,B 0,C 180,E1 -29652.376,E2 -29652.376} C_VEL
LIN {X 0,Y 56.718,Z 459.4,A -85,B 0,C 180,E1 -29658.026,E2 -29658.026} C_VEL
LIN {X 0,Y 61.803,Z 458.82,A -85,B 0,C 180,E1 -29662.749,E2 -29662.749} C_VEL
LIN {X 0,Y 67.227,Z 457.772,A -85,B 0,C 180,E1 -29666.753,E2 -29666.753} C_VEL
LIN {X 0,Y 75.965,Z 455.144,A -85,B 0,C 180,E1 -29671.509,E2 -29671.509} C_VEL
LIN {X 0,Y 85.143,Z 451.282,A -85,B 0,C 180,E1 -29675.225,E2 -29675.225} C_VEL
LIN {X 0,Y 95.36,Z 445.635,A -85,B 0,C 180,E1 -29678.363,E2 -29678.363} C_VEL
LIN {X 0,Y 104.359,Z 439.249,A -85,B 0,C 180,E1 -29680.53,E2 -29680.53} C_VEL
LIN {X 0,Y 112.612,Z 431.827,A -85,B 0,C 180,E1 -29682.124,E2 -29682.124} C_VEL
LIN {X 0,Y 119.292,Z 424.528,A -85,B 0,C 180,E1 -29683.205,E2 -29683.205} C_VEL
LIN {X 0,Y 125.085,Z 416.883,A -85,B 0,C 180,E1 -29684.008,E2 -29684.008} C_VEL
LIN {X 0,Y 128.847,Z 411.048,A -85,B 0,C 180,E1 -29684.457,E2 -29684.457} C_VEL
LIN {X 0,Y 129.789,Z 409.093,A -85,B 0,C 180,E1 -29685.086,E2 -29685.086} C_VEL
LIN {X 0,Y 129.856,Z 406.923,A -85,B 0,C 180,E1 -29690.646,E2 -29690.646} C_VEL
LIN {X 0,Y 130.006,Z 406.473,A -85,B 0,C 180,E1 -29693.783,E2 -29693.783} C_VEL
LIN {X 0,Y 129.261,Z 409.272,A -85,B 0,C 180,E1 -29699.601,E2 -29699.601} C_VEL
LIN {X 0,Y 125.579,Z 415.096,A -85,B 0,C 180,E1 -29700.32,E2 -29700.32} C_VEL
LIN {X 0,Y 120.38,Z 422.043,A -85,B 0,C 180,E1 -29701.202,E2 -29701.202} C_VEL
LIN {X 0,Y 114.303,Z 428.839,A -85,B 0,C 180,E1 -29702.382,E2 -29702.382} C_VEL
LIN {X 0,Y 107.197,Z 435.428,A -85,B 0,C 180,E1 -29703.928,E2 -29703.928} C_VEL
LIN {X 0,Y 98.934,Z 441.703,A -85,B 0,C 180,E1 -29706.008,E2 -29706.008} C_VEL
LIN {X 0,Y 90.269,Z 446.858,A -85,B 0,C 180,E1 -29708.611,E2 -29708.611} C_VEL
LIN {X 0,Y 85.246,Z 449.315,A -85,B 0,C 180,E1 -29709.908,E2 -29709.908} C_VEL
LIN {X 0,Y 76.099,Z 452.647,A -85,B 0,C 180,E1 -29711.283,E2 -29711.283} C_VEL
LIN {X 0,Y 66.77,Z 455.091,A -85,B 0,C 180,E1 -29713.143,E2 -29713.143} C_VEL
LIN {X 0,Y 61.573,Z 455.973,A -85,B 0,C 180,E1 -29715.49,E2 -29715.49} C_VEL
LIN {X 0,Y 53.078,Z 456.759,A -85,B 0,C 180,E1 -29722.052,E2 -29722.052} C_VEL
LIN {X 0,Y 47.706,Z 456.608,A -85,B 0,C 180,E1 -29727.885,E2 -29727.885} C_VEL
LIN {X 0,Y 42.931,Z 455.944,A -85,B 0,C 180,E1 -29735.066,E2 -29735.066} C_VEL
LIN {X 0,Y 37.437,Z 453.924,A -85,B 0,C 180,E1 -29748.615,E2 -29748.615} C_VEL
LIN {X 0,Y 35.072,Z 451.807,A -85,B 0,C 180,E1 -29759.938,E2 -29759.938} C_VEL
LIN {X 0,Y 34.235,Z 447.539,A -85,B 0,C 180,E1 -29778.156,E2 -29778.156} C_VEL
LIN {X 0,Y 36.556,Z 441.76,A -85,B 0,C 180,E1 -29795.518,E2 -29795.518} C_VEL
LIN {X 0,Y 40.332,Z 435.433,A -85,B 0,C 180,E1 -29807.757,E2 -29807.757} C_VEL
LIN {X 0,Y 44.204,Z 429.28,A -85,B 0,C 180,E1 -29815.929,E2 -29815.929} C_VEL
LIN {X 0,Y 48.826,Z 421.771,A -85,B 0,C 180,E1 -29822.67,E2 -29822.67} C_VEL
LIN {X 0,Y 52.982,Z 414.3,A -85,B 0,C 180,E1 -29827.304,E2 -29827.304} C_VEL
LIN {X 0,Y 56.629,Z 406.758,A -85,B 0,C 180,E1 -29830.661,E2 -29830.661} C_VEL
LIN {X 0,Y 60.091,Z 398.207,A -85,B 0,C 180,E1 -29833.404,E2 -29833.404} C_VEL
LIN {X 0,Y 63.044,Z 389.087,A -85,B 0,C 180,E1 -29835.447,E2 -29835.447} C_VEL
LIN {X 0,Y 65.764,Z 377.297,A -85,B 0,C 180,E1 -29837.219,E2 -29837.219} C_VEL
LIN {X 0,Y 67.903,Z 359.531,A -85,B 0,C 180,E1 -29838.537,E2 -29838.537} C_VEL
LIN {X 0,Y 67.988,Z 357.2,A -85,B 0,C 180,E1 -29838.891,E2 -29838.891} C_VEL
LIN {X 0,Y 65.868,Z 351.829,A -85,B 0,C 180,E1 -29843.226,E2 -29843.226} C_VEL
LIN {X 0,Y 63.687,Z 347.277,A -85,B 0,C 180,E1 -29848.569,E2 -29848.569} C_VEL
LIN {X 0,Y 61.819,Z 343.709,A -85,B 0,C 180,E1 -29854.7,E2 -29854.7} C_VEL
LIN {X 0,Y 60.285,Z 339.873,A -85,B 0,C 180,E1 -29864.023,E2 -29864.023} C_VEL
LIN {X 0,Y 60.468,Z 337.293,A -85,B 0,C 180,E1 -29877.143,E2 -29877.143} C_VEL
LIN {X 0,Y 61.13,Z 336.313,A -85,B 0,C 180,E1 -29880.922,E2 -29880.922} C_VEL
LIN {X 0,Y 61.19,Z 342.228,A -85,B 0,C 180,E1 -29884.744,E2 -29884.744} C_VEL
LIN {X 0,Y 61.799,Z 346.206,A -85,B 0,C 180,E1 -29888.605,E2 -29888.605} C_VEL
LIN {X 0,Y 62.334,Z 347.453,A -85,B 0,C 180,E1 -29890.578,E2 -29890.578} C_VEL
LIN {X 0,Y 63.657,Z 375.336,A -85,B 0,C 180,E1 -29901.26,E2 -29901.26} C_VEL
LIN {X 0,Y 64.28,Z 384.813,A -85,B 0,C 180,E1 -29905.521,E2 -29905.521} C_VEL
LIN {X 0,Y 65.034,Z 391.774,A -85,B 0,C 180,E1 -29909.474,E2 -29909.474} C_VEL
LIN {X 0,Y 66.643,Z 400.145,A -85,B 0,C 180,E1 -29915.299,E2 -29915.299} C_VEL
LIN {X 0,Y 67.763,Z 404.236,A -85,B 0,C 180,E1 -29918.506,E2 -29918.506} C_VEL
LIN {X 0,Y 67.928,Z 405.869,A -85,B 0,C 180,E1 -29919.502,E2 -29919.502} C_VEL
LIN {X 0,Y 61.101,Z 414.873,A -85,B 0,C 180,E1 -29920.355,E2 -29920.355} C_VEL
LIN {X 0,Y 54.98,Z 422.686,A -85,B 0,C 180,E1 -29922.69,E2 -29922.69} C_VEL
LIN {X 0,Y 48.964,Z 430.088,A -85,B 0,C 180,E1 -29926.957,E2 -29926.957} C_VEL
LIN {X 0,Y 43.858,Z 436.389,A -85,B 0,C 180,E1 -29933.062,E2 -29933.062} C_VEL
LIN {X 0,Y 39.786,Z 441.674,A -85,B 0,C 180,E1 -29940.935,E2 -29940.935} C_VEL
LIN {X 0,Y 36.27,Z 447.055,A -85,B 0,C 180,E1 -29953.101,E2 -29953.101} C_VEL
LIN {X 0,Y 34.994,Z 452.092,A -85,B 0,C 180,E1 -29969.998,E2 -29969.998} C_VEL
LIN {X 0,Y 35.105,Z 454.558,A -85,B 0,C 180,E1 -29981.546,E2 -29981.546} C_VEL
LIN {X 0,Y 36.461,Z 456.487,A -85,B 0,C 180,E1 -29992.673,E2 -29992.673} C_VEL
LIN {X 0,Y 39.088,Z 457.933,A -85,B 0,C 180,E1 -30002.64,E2 -30002.64} C_VEL
LIN {X 0,Y 42.719,Z 458.803,A -85,B 0,C 180,E1 -30011.15,E2 -30011.15} C_VEL
LIN {X 0,Y 47.124,Z 459.172,A -85,B 0,C 180,E1 -30018.216,E2 -30018.216} C_VEL
LIN {X 0,Y 52.243,Z 459.12,A -85,B 0,C 180,E1 -30023.816,E2 -30023.816} C_VEL
LIN {X 0,Y 57.786,Z 458.633,A -85,B 0,C 180,E1 -30028.357,E2 -30028.357} C_VEL
LIN {X 0,Y 63.607,Z 457.612,A -85,B 0,C 180,E1 -30032.117,E2 -30032.117} C_VEL
LIN {X 0,Y 72.852,Z 455.145,A -85,B 0,C 180,E1 -30036.411,E2 -30036.411} C_VEL
LIN {X 0,Y 82.422,Z 451.394,A -85,B 0,C 180,E1 -30039.709,E2 -30039.709} C_VEL
LIN {X 0,Y 91.827,Z 446.535,A -85,B 0,C 180,E1 -30042.159,E2 -30042.159} C_VEL
LIN {X 0,Y 98.858,Z 442.026,A -85,B 0,C 180,E1 -30043.684,E2 -30043.684} C_VEL
LIN {X 0,Y 105.587,Z 436.913,A -85,B 0,C 180,E1 -30044.824,E2 -30044.824} C_VEL
LIN {X 0,Y 112.339,Z 430.785,A -85,B 0,C 180,E1 -30045.855,E2 -30045.855} C_VEL
LIN {X 0,Y 118.303,Z 424.358,A -85,B 0,C 180,E1 -30046.599,E2 -30046.599} C_VEL
LIN {X 0,Y 124.079,Z 416.898,A -85,B 0,C 180,E1 -30047.239,E2 -30047.239} C_VEL
LIN {X 0,Y 125.587,Z 414.744,A -85,B 0,C 180,E1 -30047.382,E2 -30047.382} C_VEL
LIN {X 0,Y 125.989,Z 413.983,A -85,B 0,C 180,E1 -30047.999,E2 -30047.999} C_VEL
LIN {X 0,Y 126.151,Z 413.175,A -85,B 0,C 180,E1 -30050.369,E2 -30050.369} C_VEL
LIN {X 0,Y 126.341,Z 412.633,A -85,B 0,C 180,E1 -30053.602,E2 -30053.602} C_VEL
LIN {X 0,Y 125.684,Z 413.922,A -85,B 0,C 180,E1 -30056.784,E2 -30056.784} C_VEL
LIN {X 0,Y 123.88,Z 416.536,A -85,B 0,C 180,E1 -30057.2,E2 -30057.2} C_VEL
LIN {X 0,Y 116.895,Z 425.313,A -85,B 0,C 180,E1 -30058.238,E2 -30058.238} C_VEL
LIN {X 0,Y 109.109,Z 433.048,A -85,B 0,C 180,E1 -30059.551,E2 -30059.551} C_VEL
LIN {X 0,Y 101.919,Z 438.863,A -85,B 0,C 180,E1 -30060.964,E2 -30060.964} C_VEL
LIN {X 0,Y 94.965,Z 443.549,A -85,B 0,C 180,E1 -30062.465,E2 -30062.465} C_VEL
LIN {X 0,Y 86.818,Z 447.999,A -85,B 0,C 180,E1 -30064.628,E2 -30064.628} C_VEL
LIN {X 0,Y 77.975,Z 451.737,A -85,B 0,C 180,E1 -30067.508,E2 -30067.508} C_VEL
LIN {X 0,Y 67.761,Z 454.804,A -85,B 0,C 180,E1 -30071.952,E2 -30071.952} C_VEL
LIN {X 0,Y 61.573,Z 455.973,A -85,B 0,C 180,E1 -30075.49,E2 -30075.49} C_VEL
LIN {X 0,Y 56.438,Z 456.641,A -85,B 0,C 180,E1 -30078.299,E2 -30078.299} C_VEL
LIN {X 0,Y 47.241,Z 457.041,A -85,B 0,C 180,E1 -30082.477,E2 -30082.477} C_VEL
LIN {X 0,Y 38.421,Z 456.39,A -85,B 0,C 180,E1 -30088.523,E2 -30088.523} C_VEL
LIN {X 0,Y 34.192,Z 455.335,A -85,B 0,C 180,E1 -30094.83,E2 -30094.83} C_VEL
LIN {X 0,Y 28.888,Z 452.52,A -85,B 0,C 180,E1 -30112.543,E2 -30112.543} C_VEL
LIN {X 0,Y 27.217,Z 449.964,A -85,B 0,C 180,E1 -30127.215,E2 -30127.215} C_VEL
LIN {X 0,Y 27.373,Z 446.738,A -85,B 0,C 180,E1 -30142.627,E2 -30142.627} C_VEL
LIN {X 0,Y 29.978,Z 441.633,A -85,B 0,C 180,E1 -30160.13,E2 -30160.13} C_VEL
LIN {X 0,Y 34.505,Z 435.205,A -85,B 0,C 180,E1 -30174.042,E2 -30174.042} C_VEL
LIN {X 0,Y 39.053,Z 428.937,A -85,B 0,C 180,E1 -30182.678,E2 -30182.678} C_VEL
LIN {X 0,Y 43.612,Z 422.337,A -85,B 0,C 180,E1 -30188.644,E2 -30188.644} C_VEL
LIN {X 0,Y 48.256,Z 414.76,A -85,B 0,C 180,E1 -30193.305,E2 -30193.305} C_VEL
LIN {X 0,Y 52.122,Z 407.438,A -85,B 0,C 180,E1 -30196.45,E2 -30196.45} C_VEL
LIN {X 0,Y 55.853,Z 398.97,A -85,B 0,C 180,E1 -30199.026,E2 -30199.026} C_VEL
LIN {X 0,Y 58.853,Z 390.448,A -85,B 0,C 180,E1 -30200.843,E2 -30200.843} C_VEL
LIN {X 0,Y 61.587,Z 379.883,A -85,B 0,C 180,E1 -30202.403,E2 -30202.403} C_VEL
LIN {X 0,Y 63.756,Z 365.197,A -85,B 0,C 180,E1 -30203.572,E2 -30203.572} C_VEL
LIN {X 0,Y 64.259,Z 360.155,A -85,B 0,C 180,E1 -30203.947,E2 -30203.947} C_VEL
LIN {X 0,Y 62.66,Z 355.645,A -85,B 0,C 180,E1 -30208.307,E2 -30208.307} C_VEL
LIN {X 0,Y 61.243,Z 352.487,A -85,B 0,C 180,E1 -30212.92,E2 -30212.92} C_VEL
LIN {X 0,Y 60.32,Z 350.278,A -85,B 0,C 180,E1 -30216.922,E2 -30216.922} C_VEL
LIN {X 0,Y 59.169,Z 346.347,A -85,B 0,C 180,E1 -30226.937,E2 -30226.937} C_VEL
LIN {X 0,Y 59.658,Z 344.364,A -85,B 0,C 180,E1 -30237.938,E2 -30237.938} C_VEL
LIN {X 0,Y 59.731,Z 350.024,A -85,B 0,C 180,E1 -30242.805,E2 -30242.805} C_VEL
LIN {X 0,Y 60.093,Z 352.621,A -85,B 0,C 180,E1 -30245.736,E2 -30245.736} C_VEL
LIN {X 0,Y 60.223,Z 377.61,A -85,B 0,C 180,E1 -30255.895,E2 -30255.895} C_VEL
LIN {X 0,Y 60.217,Z 388.133,A -85,B 0,C 180,E1 -30261.124,E2 -30261.124} C_VEL
LIN {X 0,Y 60.504,Z 396.736,A -85,B 0,C 180,E1 -30266.773,E2 -30266.773} C_VEL
LIN {X 0,Y 61.926,Z 406.19,A -85,B 0,C 180,E1 -30274.597,E2 -30274.597} C_VEL
LIN {X 0,Y 55.007,Z 415.474,A -85,B 0,C 180,E1 -30275.459,E2 -30275.459} C_VEL
LIN {X 0,Y 48.886,Z 423.14,A -85,B 0,C 180,E1 -30277.747,E2 -30277.747} C_VEL
LIN {X 0,Y 42.673,Z 430.399,A -85,B 0,C 180,E1 -30282.027,E2 -30282.027} C_VEL
LIN {X 0,Y 37.232,Z 436.634,A -85,B 0,C 180,E1 -30288.639,E2 -30288.639} C_VEL
LIN {X 0,Y 32.798,Z 441.824,A -85,B 0,C 180,E1 -30297.606,E2 -30297.606} C_VEL
LIN {X 0,Y 29.603,Z 446.181,A -85,B 0,C 180,E1 -30309.135,E2 -30309.135} C_VEL
LIN {X 0,Y 27.919,Z 451.328,A -85,B 0,C 180,E1 -30329.997,E2 -30329.997} C_VEL
LIN {X 0,Y 28.194,Z 453.898,A -85,B 0,C 180,E1 -30344.432,E2 -30344.432} C_VEL
LIN {X 0,Y 30.051,Z 455.927,A -85,B 0,C 180,E1 -30357.884,E2 -30357.884} C_VEL
LIN {X 0,Y 33.33,Z 457.423,A -85,B 0,C 180,E1 -30369.238,E2 -30369.238} C_VEL
LIN {X 0,Y 37.665,Z 458.336,A -85,B 0,C 180,E1 -30378.274,E2 -30378.274} C_VEL
LIN {X 0,Y 42.716,Z 458.798,A -85,B 0,C 180,E1 -30385.347,E2 -30385.347} C_VEL
LIN {X 0,Y 48.385,Z 458.839,A -85,B 0,C 180,E1 -30390.632,E2 -30390.632} C_VEL
LIN {X 0,Y 54.393,Z 458.422,A -85,B 0,C 180,E1 -30394.746,E2 -30394.746} C_VEL
LIN {X 0,Y 60.611,Z 457.425,A -85,B 0,C 180,E1 -30398.065,E2 -30398.065} C_VEL
LIN {X 0,Y 67.048,Z 455.949,A -85,B 0,C 180,E1 -30400.623,E2 -30400.623} C_VEL
LIN {X 0,Y 76.908,Z 452.819,A -85,B 0,C 180,E1 -30403.635,E2 -30403.635} C_VEL
LIN {X 0,Y 86.967,Z 448.414,A -85,B 0,C 180,E1 -30405.867,E2 -30405.867} C_VEL
LIN {X 0,Y 97.107,Z 442.378,A -85,B 0,C 180,E1 -30407.695,E2 -30407.695} C_VEL
LIN {X 0,Y 103.958,Z 437.406,A -85,B 0,C 180,E1 -30408.593,E2 -30408.593} C_VEL
LIN {X 0,Y 110.826,Z 431.44,A -85,B 0,C 180,E1 -30409.393,E2 -30409.393} C_VEL
LIN {X 0,Y 117.731,Z 424.191,A -85,B 0,C 180,E1 -30410.051,E2 -30410.051} C_VEL
LIN {X 0,Y 121.19,Z 420.086,A -85,B 0,C 180,E1 -30410.35,E2 -30410.35} C_VEL
LIN {X 0,Y 122.198,Z 418.464,A -85,B 0,C 180,E1 -30413.384,E2 -30413.384} C_VEL
LIN {X 0,Y 122.071,Z 418.654,A -85,B 0,C 180,E1 -30413.875,E2 -30413.875} C_VEL
LIN {X 0,Y 120.073,Z 421.155,A -85,B 0,C 180,E1 -30414.279,E2 -30414.279} C_VEL
LIN {X 0,Y 112.845,Z 429.09,A -85,B 0,C 180,E1 -30415.186,E2 -30415.186} C_VEL
LIN {X 0,Y 105.648,Z 435.556,A -85,B 0,C 180,E1 -30416.222,E2 -30416.222} C_VEL
LIN {X 0,Y 98.493,Z 440.872,A -85,B 0,C 180,E1 -30417.391,E2 -30417.391} C_VEL
LIN {X 0,Y 91.388,Z 445.244,A -85,B 0,C 180,E1 -30418.654,E2 -30418.654} C_VEL
LIN {X 0,Y 84.335,Z 448.826,A -85,B 0,C 180,E1 -30420.207,E2 -30420.207} C_VEL
LIN {X 0,Y 73.899,Z 452.881,A -85,B 0,C 180,E1 -30423.071,E2 -30423.071} C_VEL
LIN {X 0,Y 63.707,Z 455.583,A -85,B 0,C 180,E1 -30426.858,E2 -30426.858} C_VEL
LIN {X 0,Y 57.11,Z 456.583,A -85,B 0,C 180,E1 -30430.112,E2 -30430.112} C_VEL
LIN {X 0,Y 46.742,Z 457.138,A -85,B 0,C 180,E1 -30437.471,E2 -30437.471} C_VEL
LIN {X 0,Y 39.116,Z 456.444,A -85,B 0,C 180,E1 -30446.061,E2 -30446.061} C_VEL
LIN {X 0,Y 34.192,Z 455.335,A -85,B 0,C 180,E1 -30454.83,E2 -30454.83} C_VEL
LIN {X 0,Y 30.502,Z 454.048,A -85,B 0,C 180,E1 -30462.629,E2 -30462.629} C_VEL
LIN {X 0,Y 24.348,Z 451.26,A -85,B 0,C 180,E1 -30477.942,E2 -30477.942} C_VEL
LIN {X 0,Y 21.057,Z 448.365,A -85,B 0,C 180,E1 -30494.957,E2 -30494.957} C_VEL
LIN {X 0,Y 20.791,Z 445.795,A -85,B 0,C 180,E1 -30509.67,E2 -30509.67} C_VEL
LIN {X 0,Y 21.243,Z 444.816,A -85,B 0,C 180,E1 -30514.284,E2 -30514.284} C_VEL
LIN {X 0,Y 25.765,Z 439.063,A -85,B 0,C 180,E1 -30534.155,E2 -30534.155} C_VEL
LIN {X 0,Y 31.842,Z 432.039,A -85,B 0,C 180,E1 -30547.374,E2 -30547.374} C_VEL
LIN {X 0,Y 38.235,Z 423.951,A -85,B 0,C 180,E1 -30555.422,E2 -30555.422} C_VEL
LIN {X 0,Y 43.065,Z 417.028,A -85,B 0,C 180,E1 -30559.637,E2 -30559.637} C_VEL
LIN {X 0,Y 48.244,Z 408.118,A -85,B 0,C 180,E1 -30563.249,E2 -30563.249} C_VEL
LIN {X 0,Y 51.918,Z 400.501,A -85,B 0,C 180,E1 -30565.31,E2 -30565.31} C_VEL
LIN {X 0,Y 55.239,Z 391.86,A -85,B 0,C 180,E1 -30567.003,E2 -30567.003} C_VEL
LIN {X 0,Y 57.856,Z 382.809,A -85,B 0,C 180,E1 -30568.249,E2 -30568.249} C_VEL
LIN {X 0,Y 59.735,Z 373.526,A -85,B 0,C 180,E1 -30568.993,E2 -30568.993} C_VEL
LIN {X 0,Y 61.009,Z 363.032,A -85,B 0,C 180,E1 -30569.794,E2 -30569.794} C_VEL
LIN {X 0,Y 59.797,Z 359.336,A -85,B 0,C 180,E1 -30574.575,E2 -30574.575} C_VEL
LIN {X 0,Y 58.87,Z 356.714,A -85,B 0,C 180,E1 -30579.552,E2 -30579.552} C_VEL
LIN {X 0,Y 58.198,Z 353.234,A -85,B 0,C 180,E1 -30588.706,E2 -30588.706} C_VEL
LIN {X 0,Y 58.415,Z 352.191,A -85,B 0,C 180,E1 -30595.304,E2 -30595.304} C_VEL
LIN {X 0,Y 58.355,Z 356.968,A -85,B 0,C 180,E1 -30600.165,E2 -30600.165} C_VEL
LIN {X 0,Y 57.456,Z 377.887,A -85,B 0,C 180,E1 -30609.084,E2 -30609.084} C_VEL
LIN {X 0,Y 56.676,Z 388.374,A -85,B 0,C 180,E1 -30614.383,E2 -30614.383} C_VEL
LIN {X 0,Y 56.03,Z 397.263,A -85,B 0,C 180,E1 -30620.305,E2 -30620.305} C_VEL
LIN {X 0,Y 56.201,Z 406.958,A -85,B 0,C 180,E1 -30628.91,E2 -30628.91} C_VEL
LIN {X 0,Y 49.471,Z 416.044,A -85,B 0,C 180,E1 -30629.523,E2 -30629.523} C_VEL
LIN {X 0,Y 43.267,Z 423.597,A -85,B 0,C 180,E1 -30631.482,E2 -30631.482} C_VEL
LIN {X 0,Y 38.22,Z 429.262,A -85,B 0,C 180,E1 -30634.398,E2 -30634.398} C_VEL
LIN {X 0,Y 32.315,Z 435.501,A -85,B 0,C 180,E1 -30640.418,E2 -30640.418} C_VEL
LIN {X 0,Y 27.125,Z 440.827,A -85,B 0,C 180,E1 -30649.625,E2 -30649.625} C_VEL
LIN {X 0,Y 23.163,Z 445.307,A -85,B 0,C 180,E1 -30662.924,E2 -30662.924} C_VEL
LIN {X 0,Y 21.05,Z 449.044,A -85,B 0,C 180,E1 -30680.387,E2 -30680.387} C_VEL
LIN {X 0,Y 20.897,Z 452.024,A -85,B 0,C 180,E1 -30699.677,E2 -30699.677} C_VEL
LIN {X 0,Y 24.004,Z 455.357,A -85,B 0,C 180,E1 -30725.839,E2 -30725.839} C_VEL
LIN {X 0,Y 28.184,Z 456.87,A -85,B 0,C 180,E1 -30738.419,E2 -30738.419} C_VEL
LIN {X 0,Y 33.355,Z 457.868,A -85,B 0,C 180,E1 -30747.435,E2 -30747.435} C_VEL
LIN {X 0,Y 39.112,Z 458.424,A -85,B 0,C 180,E1 -30753.949,E2 -30753.949} C_VEL
LIN {X 0,Y 45.323,Z 458.558,A -85,B 0,C 180,E1 -30758.49,E2 -30758.49} C_VEL
LIN {X 0,Y 51.758,Z 458.169,A -85,B 0,C 180,E1 -30761.893,E2 -30761.893} C_VEL
LIN {X 0,Y 58.331,Z 457.237,A -85,B 0,C 180,E1 -30764.548,E2 -30764.548} C_VEL
LIN {X 0,Y 65.042,Z 455.856,A -85,B 0,C 180,E1 -30766.521,E2 -30766.521} C_VEL
LIN {X 0,Y 75.216,Z 452.826,A -85,B 0,C 180,E1 -30768.837,E2 -30768.837} C_VEL
LIN {X 0,Y 85.513,Z 448.555,A -85,B 0,C 180,E1 -30770.478,E2 -30770.478} C_VEL
LIN {X 0,Y 95.848,Z 442.73,A -85,B 0,C 180,E1 -30771.836,E2 -30771.836} C_VEL
LIN {X 0,Y 99.319,Z 440.374,A -85,B 0,C 180,E1 -30772.162,E2 -30772.162} C_VEL
LIN {X 0,Y 99.112,Z 440.455,A -85,B 0,C 180,E1 -30773.086,E2 -30773.086} C_VEL
LIN {X 0,Y 91.86,Z 444.969,A -85,B 0,C 180,E1 -30774.038,E2 -30774.038} C_VEL
LIN {X 0,Y 84.377,Z 448.789,A -85,B 0,C 180,E1 -30775.207,E2 -30775.207} C_VEL
LIN {X 0,Y 73.876,Z 452.85,A -85,B 0,C 180,E1 -30777.277,E2 -30777.277} C_VEL
LIN {X 0,Y 70.316,Z 454.005,A -85,B 0,C 180,E1 -30778.13,E2 -30778.13} C_VEL
LIN {X 0,Y 63.251,Z 455.671,A -85,B 0,C 180,E1 -30780.14,E2 -30780.14} C_VEL
LIN {X 0,Y 56.28,Z 456.771,A -85,B 0,C 180,E1 -30782.592,E2 -30782.592} C_VEL
LIN {X 0,Y 43.811,Z 457.46,A -85,B 0,C 180,E1 -30789.201,E2 -30789.201} C_VEL
LIN {X 0,Y 36.459,Z 456.939,A -85,B 0,C 180,E1 -30795.469,E2 -30795.469} C_VEL
LIN {X 0,Y 28.827,Z 455.348,A -85,B 0,C 180,E1 -30806.354,E2 -30806.354} C_VEL
LIN {X 0,Y 23.423,Z 453.235,A -85,B 0,C 180,E1 -30821.403,E2 -30821.403} C_VEL
LIN {X 0,Y 20.584,Z 450.761,A -85,B 0,C 180,E1 -30839.197,E2 -30839.197} C_VEL
LIN {X 0,Y 20.744,Z 445.718,A -85,B 0,C 180,E1 -30870.004,E2 -30870.004} C_VEL
LIN {X 0,Y 21.243,Z 444.816,A -85,B 0,C 180,E1 -30874.284,E2 -30874.284} C_VEL
LIN {X 0,Y 22.814,Z 441.875,A -85,B 0,C 180,E1 -30886.979,E2 -30886.979} C_VEL
LIN {X 0,Y 24.356,Z 438.663,A -85,B 0,C 180,E1 -30898.684,E2 -30898.684} C_VEL
LIN {X 0,Y 29.304,Z 430.885,A -85,B 0,C 180,E1 -30918.383,E2 -30918.383} C_VEL
LIN {X 0,Y 31.996,Z 427.438,A -85,B 0,C 180,E1 -30922.773,E2 -30922.773} C_VEL
LIN {X 0,Y 33.18,Z 425.983,A -85,B 0,C 180,E1 -30923.915,E2 -30923.915} C_VEL
LIN {X 0,Y 39.493,Z 417.831,A -85,B 0,C 180,E1 -30928.19,E2 -30928.19} C_VEL
LIN {X 0,Y 44.495,Z 409.992,A -85,B 0,C 180,E1 -30930.817,E2 -30930.817} C_VEL
LIN {X 0,Y 48.855,Z 401.688,A -85,B 0,C 180,E1 -30932.589,E2 -30932.589} C_VEL
LIN {X 0,Y 52.308,Z 393.403,A -85,B 0,C 180,E1 -30933.893,E2 -30933.893} C_VEL
LIN {X 0,Y 55.301,Z 383.854,A -85,B 0,C 180,E1 -30934.913,E2 -30934.913} C_VEL
LIN {X 0,Y 57.223,Z 375.074,A -85,B 0,C 180,E1 -30935.512,E2 -30935.512} C_VEL
LIN {X 0,Y 58.414,Z 366.495,A -85,B 0,C 180,E1 -30936.115,E2 -30936.115} C_VEL
LIN {X 0,Y 57.556,Z 363.183,A -85,B 0,C 180,E1 -30942.25,E2 -30942.25} C_VEL
LIN {X 0,Y 57.29,Z 360.013,A -85,B 0,C 180,E1 -30951.114,E2 -30951.114} C_VEL
LIN {X 0,Y 57.336,Z 359.82,A -85,B 0,C 180,E1 -30952.982,E2 -30952.982} C_VEL
LIN {X 0,Y 57.226,Z 361.096,A -85,B 0,C 180,E1 -30954.313,E2 -30954.313} C_VEL
LIN {X 0,Y 55.534,Z 378.578,A -85,B 0,C 180,E1 -30961.877,E2 -30961.877} C_VEL
LIN {X 0,Y 53.821,Z 389.649,A -85,B 0,C 180,E1 -30967.527,E2 -30967.527} C_VEL
LIN {X 0,Y 52.217,Z 398.712,A -85,B 0,C 180,E1 -30973.693,E2 -30973.693} C_VEL
LIN {X 0,Y 51.251,Z 406.778,A -85,B 0,C 180,E1 -30981.127,E2 -30981.127} C_VEL
LIN {X 0,Y 50.733,Z 408.511,A -85,B 0,C 180,E1 -30982.353,E2 -30982.353} C_VEL
LIN {X 0,Y 45.553,Z 415.494,A -85,B 0,C 180,E1 -30982.223,E2 -30982.223} C_VEL
LIN {X 0,Y 40.084,Z 422.121,A -85,B 0,C 180,E1 -30982.997,E2 -30982.997} C_VEL
LIN {X 0,Y 32.918,Z 429.745,A -85,B 0,C 180,E1 -30985.827,E2 -30985.827} C_VEL
LIN {X 0,Y 26.713,Z 435.752,A -85,B 0,C 180,E1 -30991.223,E2 -30991.223} C_VEL
LIN {X 0,Y 20.849,Z 440.978,A -85,B 0,C 180,E1 -31000.667,E2 -31000.667} C_VEL
LIN {X 0,Y 15.325,Z 446.317,A -85,B 0,C 180,E1 -31022.698,E2 -31022.698} C_VEL
LIN {X 0,Y 13.8,Z 449.802,A -85,B 0,C 180,E1 -31049.994,E2 -31049.994} C_VEL
LIN {X 0,Y 16.566,Z 453.669,A -85,B 0,C 180,E1 -31089.514,E2 -31089.514} C_VEL
LIN {X 0,Y 24.065,Z 456.308,A -85,B 0,C 180,E1 -31111.174,E2 -31111.174} C_VEL
LIN {X 0,Y 30.13,Z 457.401,A -85,B 0,C 180,E1 -31118.903,E2 -31118.903} C_VEL
LIN {X 0,Y 36.552,Z 458.05,A -85,B 0,C 180,E1 -31124.013,E2 -31124.013} C_VEL
LIN {X 0,Y 43.226,Z 458.258,A -85,B 0,C 180,E1 -31127.289,E2 -31127.289} C_VEL
LIN {X 0,Y 50.005,Z 457.888,A -85,B 0,C 180,E1 -31129.668,E2 -31129.668} C_VEL
LIN {X 0,Y 56.853,Z 457.05,A -85,B 0,C 180,E1 -31131.459,E2 -31131.459} C_VEL
LIN {X 0,Y 63.764,Z 455.764,A -85,B 0,C 180,E1 -31132.723,E2 -31132.723} C_VEL
LIN {X 0,Y 63.674,Z 455.754,A -85,B 0,C 180,E1 -31133.393,E2 -31133.393} C_VEL
LIN {X 0,Y 56.436,Z 456.957,A -85,B 0,C 180,E1 -31135.017,E2 -31135.017} C_VEL
LIN {X 0,Y 49.259,Z 457.635,A -85,B 0,C 180,E1 -31137.061,E2 -31137.061} C_VEL
LIN {X 0,Y 41.939,Z 457.782,A -85,B 0,C 180,E1 -31139.969,E2 -31139.969} C_VEL
LIN {X 0,Y 35.211,Z 457.391,A -85,B 0,C 180,E1 -31143.664,E2 -31143.664} C_VEL
LIN {X 0,Y 28.482,Z 456.379,A -85,B 0,C 180,E1 -31149.267,E2 -31149.267} C_VEL
LIN {X 0,Y 19.21,Z 453.882,A -85,B 0,C 180,E1 -31164.913,E2 -31164.913} C_VEL
LIN {X 0,Y 13.33,Z 450.023,A -85,B 0,C 180,E1 -31198.187,E2 -31198.187} C_VEL
LIN {X 0,Y 14.745,Z 444.714,A -85,B 0,C 180,E1 -31243.46,E2 -31243.46} C_VEL
LIN {X 0,Y 20.702,Z 438.925,A -85,B 0,C 180,E1 -31266.453,E2 -31266.453} C_VEL
LIN {X 0,Y 28,Z 431.738,A -85,B 0,C 180,E1 -31278.856,E2 -31278.856} C_VEL
LIN {X 0,Y 33.18,Z 425.983,A -85,B 0,C 180,E1 -31283.915,E2 -31283.915} C_VEL
LIN {X 0,Y 36.449,Z 421.637,A -85,B 0,C 180,E1 -31287.397,E2 -31287.397} C_VEL
LIN {X 0,Y 40.974,Z 414.033,A -85,B 0,C 180,E1 -31294.125,E2 -31294.125} C_VEL
LIN {X 0,Y 45.184,Z 405.994,A -85,B 0,C 180,E1 -31299.454,E2 -31299.454} C_VEL
LIN {X 0,Y 47.682,Z 400.681,A -85,B 0,C 180,E1 -31300.964,E2 -31300.964} C_VEL
LIN {X 0,Y 51.227,Z 392.125,A -85,B 0,C 180,E1 -31301.674,E2 -31301.674} C_VEL
LIN {X 0,Y 54.012,Z 383.132,A -85,B 0,C 180,E1 -31302.275,E2 -31302.275} C_VEL
LIN {X 0,Y 56.037,Z 373.572,A -85,B 0,C 180,E1 -31302.579,E2 -31302.579} C_VEL
LIN {X 0,Y 56.509,Z 370.594,A -85,B 0,C 180,E1 -31302.876,E2 -31302.876} C_VEL
LIN {X 0,Y 56.296,Z 368.238,A -85,B 0,C 180,E1 -31308.936,E2 -31308.936} C_VEL
LIN {X 0,Y 56.23,Z 368.596,A -85,B 0,C 180,E1 -31309.625,E2 -31309.625} C_VEL
LIN {X 0,Y 53.98,Z 381.691,A -85,B 0,C 180,E1 -31315.391,E2 -31315.391} C_VEL
LIN {X 0,Y 51.745,Z 390.931,A -85,B 0,C 180,E1 -31320.025,E2 -31320.025} C_VEL
LIN {X 0,Y 49.431,Z 399.288,A -85,B 0,C 180,E1 -31325.578,E2 -31325.578} C_VEL
LIN {X 0,Y 47.342,Z 407.276,A -85,B 0,C 180,E1 -31332.898,E2 -31332.898} C_VEL
LIN {X 0,Y 46.64,Z 409.216,A -85,B 0,C 180,E1 -31334.395,E2 -31334.395} C_VEL
LIN {X 0,Y 40.647,Z 417.217,A -85,B 0,C 180,E1 -31333.442,E2 -31333.442} C_VEL
LIN {X 0,Y 33.911,Z 424.973,A -85,B 0,C 180,E1 -31333.487,E2 -31333.487} C_VEL
LIN {X 0,Y 26.773,Z 432.034,A -85,B 0,C 180,E1 -31335.268,E2 -31335.268} C_VEL
LIN {X 0,Y 17.12,Z 439.981,A -85,B 0,C 180,E1 -31342.52,E2 -31342.52} C_VEL
LIN {X 0,Y 9.626,Z 445.443,A -85,B 0,C 180,E1 -31363.093,E2 -31363.093} C_VEL
LIN {X 0,Y 6.753,Z 449.04,A -85,B 0,C 180,E1 -31409.988,E2 -31409.988} C_VEL
LIN {X 0,Y 9.299,Z 451.904,A -85,B 0,C 180,E1 -31459.084,E2 -31459.084} C_VEL
LIN {X 0,Y 15.013,Z 454.093,A -85,B 0,C 180,E1 -31479.412,E2 -31479.412} C_VEL
LIN {X 0,Y 21.559,Z 455.747,A -85,B 0,C 180,E1 -31487.933,E2 -31487.933} C_VEL
LIN {X 0,Y 28.359,Z 456.934,A -85,B 0,C 180,E1 -31492.415,E2 -31492.415} C_VEL
LIN {X 0,Y 28.258,Z 456.877,A -85,B 0,C 180,E1 -31494.15,E2 -31494.15} C_VEL
LIN {X 0,Y 19.491,Z 455.038,A -85,B 0,C 180,E1 -31499.934,E2 -31499.934} C_VEL
LIN {X 0,Y 10.917,Z 452.21,A -85,B 0,C 180,E1 -31515.085,E2 -31515.085} C_VEL
LIN {X 0,Y 5.993,Z 447.607,A -85,B 0,C 180,E1 -31590.013,E2 -31590.013} C_VEL
LIN {X 0,Y 12.181,Z 442.447,A -85,B 0,C 180,E1 -31636.165,E2 -31636.165} C_VEL
LIN {X 0,Y 18.802,Z 437.423,A -85,B 0,C 180,E1 -31647.258,E2 -31647.258} C_VEL
LIN {X 0,Y 25.598,Z 431.396,A -85,B 0,C 180,E1 -31653.172,E2 -31653.172} C_VEL
LIN {X 0,Y 32.551,Z 424.038,A -85,B 0,C 180,E1 -31656.586,E2 -31656.586} C_VEL
LIN {X 0,Y 38.548,Z 416.361,A -85,B 0,C 180,E1 -31658.652,E2 -31658.652} C_VEL
LIN {X 0,Y 43.355,Z 408.912,A -85,B 0,C 180,E1 -31659.988,E2 -31659.988} C_VEL
LIN {X 0,Y 47.682,Z 400.681,A -85,B 0,C 180,E1 -31660.964,E2 -31660.964} C_VEL
LIN {X 0,Y 48.033,Z 399.68,A -85,B 0,C 180,E1 -31661.965,E2 -31661.965} C_VEL
LIN {X 0,Y 47.986,Z 399.172,A -85,B 0,C 180,E1 -31664.998,E2 -31664.998} C_VEL
LIN {X 0,Y 47.421,Z 399.974,A -85,B 0,C 180,E1 -31669.619,E2 -31669.619} C_VEL
LIN {X 0,Y 46.18,Z 403.25,A -85,B 0,C 180,E1 -31676.871,E2 -31676.871} C_VEL
LIN {X 0,Y 45.047,Z 406.606,A -85,B 0,C 180,E1 -31682.155,E2 -31682.155} C_VEL
LIN {X 0,Y 44,Z 409.253,A -85,B 0,C 180,E1 -31685.09,E2 -31685.09} C_VEL
LIN {X 0,Y 43.866,Z 409.576,A -85,B 0,C 180,E1 -31685.391,E2 -31685.391} C_VEL
LIN {X 0,Y 38.725,Z 416.673,A -85,B 0,C 180,E1 -31683.44,E2 -31683.44} C_VEL
LIN {X 0,Y 32.755,Z 423.759,A -85,B 0,C 180,E1 -31681.641,E2 -31681.641} C_VEL
LIN {X 0,Y 26.183,Z 430.401,A -85,B 0,C 180,E1 -31680.154,E2 -31680.154} C_VEL
LIN {X 0,Y 19.331,Z 436.253,A -85,B 0,C 180,E1 -31678.976,E2 -31678.976} C_VEL
LIN {X 0,Y 12.309,Z 441.294,A -85,B 0,C 180,E1 -31677.808,E2 -31677.808} C_VEL
LIN {X 0,Y 7.057,Z 444.549,A -85,B 0,C 180,E1 -31674.907,E2 -31674.907} C_VEL
LIN {X 0,Y 17.877,Z 437.175,A -85,B 0,C 180,E1 -31669.388,E2 -31669.388} C_VEL
LIN {X 0,Y 25.038,Z 431.039,A -85,B 0,C 180,E1 -31669.257,E2 -31669.257} C_VEL
LIN {X 0,Y 32.205,Z 423.546,A -85,B 0,C 180,E1 -31669.136,E2 -31669.136} C_VEL
LIN {X 0,Y 38.164,Z 415.948,A -85,B 0,C 180,E1 -31669.239,E2 -31669.239} C_VEL
LIN {X 0,Y 42.905,Z 408.611,A -85,B 0,C 180,E1 -31669.373,E2 -31669.373} C_VEL
LIN {X 0,Y 47.014,Z 400.838,A -85,B 0,C 180,E1 -31669.522,E2 -31669.522} C_VEL
LIN {X 0,Y 50.897,Z 391.45,A -85,B 0,C 180,E1 -31669.635,E2 -31669.635} C_VEL
LIN {X 0,Y 51.362,Z 390.145,A -85,B 0,C 180,E1 -31671.028,E2 -31671.028} C_VEL
LIN {X 0,Y 47.738,Z 399.903,A -85,B 0,C 180,E1 -31676.859,E2 -31676.859} C_VEL
LIN {X 0,Y 44.979,Z 406.858,A -85,B 0,C 180,E1 -31682.64,E2 -31682.64} C_VEL
LIN {X 0,Y 44,Z 409.253,A -85,B 0,C 180,E1 -31685.09,E2 -31685.09} C_VEL
LIN {X 0,Y 43.772,Z 410.524,A -85,B 0,C 180,E1 -31685.606,E2 -31685.606} C_VEL
LIN {X 0,Y 43.772,Z 600,A -85,B 0,C 180,E1 -31685.606,E2 -31685.606} C_VEL
LIN {X 0,Y 43.772,Z 600,A -85,B 0,C 180,E1 -31685.606,E2 -31685.606}

QRS_NEXT_CUT()

QRS_NEXT()
QRS_HOME()

END
